PROGRAM F06_OuterAutomationCtrl
VAR

END_VAR

CASE gDevice.eAutomationMode OF

E_SYSTEM_EXTERNAL:
	gDevice.stMetsStatus.bUseOverlayPanel  := FALSE;

E_SYSTEM_CML:
	PRG_CML_01_InfeedCtrl();
	PRG_CML_02_LoweratorCtrl();

	gDevice.stMetsStatus.bUseOverlayPanel  := FALSE;

E_SYSTEM_LARS:
	PRG_LARS_01_TransportConvCtrl();
	PRG_LARS_02_GateSeparationCtrl();
	PRG_LARS_03_AddtitionalConvCtrl();

	gDevice.stMetsStatus.bUseOverlayPanel  := FALSE;

E_SYSTEM_SIDEFLEX:
	PRG_SFLX_01_TransportConvCtrl();
	PRG_SFLX_02_OutfeedConvCtrl();
	PRG_SFLX_03_AddtitionalConvCtrl();

	gDevice.stMetsStatus.bUseOverlayPanel  := FALSE;

ELSE
	gDevice.stMetsStatus.bUseOverlayPanel  := FALSE;

END_CASE

END_PROGRAM

(* stored: Version 1.1.0.1
   POU F06_OuterAutomationCtrl: Id {8e1209bb-c096-48ee-93e8-a1f6ef4c4533}, SpecialFunc None *)
